INTERFACE ITF_UNIT_Blikkenvullijn

METHOD Auto : BOOL
VAR_INPUT
END_VAR
END_METHOD

METHOD FB_init : BOOL
VAR_INPUT
	bInitRetains : BOOL; // if TRUE, the retain variables are initialized (warm start / cold start)
	bInCopyCode : BOOL;  // if TRUE, the instance afterwards gets moved into the copy code (online change)
END_VAR
END_METHOD

METHOD Manueel : BOOL
VAR_INPUT
END_VAR
END_METHOD

END_INTERFACE

(* stored: Version 1.1.0.1, ProductVersion 3.1.4024.12
   Itf ITF_UNIT_Blikkenvullijn: Id {b0828150-22c5-45c8-9e2c-aea04fc32620}
   Method Auto: Id {5b284624-3ca7-40d4-81f8-92598c6dc748}
   Method FB_init: Id {f09ea582-3a2e-488e-b32f-fc9d8bf63c1d}
   Method Manueel: Id {129ba574-754c-430f-99a1-b48df9bf28d1} *)
